Staubli VAL3: isStopped.pgx

public program isStopped(bool& x_bBool)
begin
  //
  if workingMode()!=4
    logMsg("机器人有报警,循环停止")
    return
  endIf

  if io:dInStop==true
    logMsg("机器人程序停止")
    return
  endIf


end
